//-----------------------			Inicia lavagem nas linhas						-----------------------//
{region "Inicio de lavagem"}
//Inicio da lavagem da linha 1
IF ComandoSalvar[84] THEN
	InsertParada(Insert:= TRUE, NomeComando:= 'INICIO LAV. L1', InsertOut=> bExecuteInsert, Comando=> sCmdInsert);
	ComandoSalvar[84] := FALSE;
END_IF	
//Inicio da lavagem da linha 2 
IF ComandoSalvar[85] THEN
	InsertParada(Insert:= TRUE, NomeComando:= 'INICIO LAV. L2', InsertOut=> bExecuteInsert, Comando=> sCmdInsert);
	ComandoSalvar[85] := FALSE;
END_IF
//Inicio da lavagem da linha 3
IF ComandoSalvar[86] THEN
	InsertParada(Insert:= TRUE, NomeComando:= 'INICIO LAV. L3', InsertOut=> bExecuteInsert, Comando=> sCmdInsert);
	ComandoSalvar[86] := FALSE;
END_IF	 
//Inicio da lavagem da linha 4
IF ComandoSalvar[87] THEN
	InsertParada(Insert:= TRUE, NomeComando:= 'INICIO LAV. L4', InsertOut=> bExecuteInsert, Comando=> sCmdInsert);
	ComandoSalvar[87] := FALSE;
END_IF	 
//Inicio da lavagem da linha 5
IF ComandoSalvar[88] THEN
	InsertParada(Insert:= TRUE, NomeComando:= 'INICIO LAV. L5', InsertOut=> bExecuteInsert, Comando=> sCmdInsert);
	ComandoSalvar[88] := FALSE;
END_IF	 
//Inicio da lavagem da linha 6
IF ComandoSalvar[89] THEN
	InsertParada(Insert:= TRUE, NomeComando:= 'INICIO LAV. L6', InsertOut=> bExecuteInsert, Comando=> sCmdInsert);
	ComandoSalvar[89] := FALSE;
END_IF	 
//Inicio da lavagem da linha 7
IF ComandoSalvar[90] THEN
	InsertParada(Insert:= TRUE, NomeComando:= 'INICIO LAV. L7', InsertOut=> bExecuteInsert, Comando=> sCmdInsert);
	ComandoSalvar[90] := FALSE;
END_IF	 
//Inicio da lavagem da linha 8
IF ComandoSalvar[91] THEN
	InsertParada(Insert:= TRUE, NomeComando:= 'INICIO LAV. L8', InsertOut=> bExecuteInsert, Comando=> sCmdInsert);
	ComandoSalvar[91] := FALSE;
END_IF
//Inicio da lavagem da linha 9
IF ComandoSalvar[92] THEN
	InsertParada(Insert:= TRUE, NomeComando:= 'INICIO LAV. L9', InsertOut=> bExecuteInsert, Comando=> sCmdInsert);
	ComandoSalvar[92] := FALSE;
END_IF 
//Inicio da lavagem da linha 10
IF ComandoSalvar[93] THEN
	InsertParada(Insert:= TRUE, NomeComando:= 'INICIO LAV. L10', InsertOut=> bExecuteInsert, Comando=> sCmdInsert);
	ComandoSalvar[93] := FALSE;
END_IF
//Inicio da lavagem da linha 11
IF ComandoSalvar[94] THEN
	InsertParada(Insert:= TRUE, NomeComando:= 'INICIO LAV. L11', InsertOut=> bExecuteInsert, Comando=> sCmdInsert);
	ComandoSalvar[94] := FALSE;
END_IF
//Inicio da lavagem da linha 12
IF ComandoSalvar[95] THEN
	InsertParada(Insert:= TRUE, NomeComando:= 'INICIO LAV. L12', InsertOut=> bExecuteInsert, Comando=> sCmdInsert);
	ComandoSalvar[95] := FALSE;
END_IF
{endregion}

//-----------------------			Para lavagem nas linhas							-----------------------//
{Region "Para a lavagem"}
//Parada da lavagem da linha 1
IF ComandoSalvar[96] THEN
	InsertParada(Insert:= TRUE, NomeComando:= 'PARA LAV. L1', InsertOut=> bExecuteInsert, Comando=> sCmdInsert);
	ComandoSalvar[96] := FALSE;
END_IF	
//Parada da lavagem da linha 2
IF ComandoSalvar[97] THEN
	InsertParada(Insert:= TRUE, NomeComando:= 'PARA LAV. L2', InsertOut=> bExecuteInsert, Comando=> sCmdInsert);
	ComandoSalvar[97] := FALSE;
END_IF	
//Parada da lavagem da linha 3
IF ComandoSalvar[98] THEN
	InsertParada(Insert:= TRUE, NomeComando:= 'PARA LAV. L3', InsertOut=> bExecuteInsert, Comando=> sCmdInsert);
	ComandoSalvar[98] := FALSE;
END_IF	
//Parada da lavagem da linha 4
IF ComandoSalvar[99] THEN
	InsertParada(Insert:= TRUE, NomeComando:= 'PARA LAV. L4', InsertOut=> bExecuteInsert, Comando=> sCmdInsert);
	ComandoSalvar[99] := FALSE;
END_IF	
//Parada da lavagem da linha 5
IF ComandoSalvar[100] THEN
	InsertParada(Insert:= TRUE, NomeComando:= 'PARA LAV. L5', InsertOut=> bExecuteInsert, Comando=> sCmdInsert);
	ComandoSalvar[100] := FALSE;
END_IF	
//Parada da lavagem da linha 6
IF ComandoSalvar[101] THEN
	InsertParada(Insert:= TRUE, NomeComando:= 'PARA LAV. L6', InsertOut=> bExecuteInsert, Comando=> sCmdInsert);
	ComandoSalvar[101] := FALSE;
END_IF	
//Parada da lavagem da linha 7
IF ComandoSalvar[102] THEN
	InsertParada(Insert:= TRUE, NomeComando:= 'PARA LAV. L7', InsertOut=> bExecuteInsert, Comando=> sCmdInsert);
	ComandoSalvar[102] := FALSE;
END_IF	
//Parada da lavagem da linha 8
IF ComandoSalvar[103] THEN
	InsertParada(Insert:= TRUE, NomeComando:= 'PARA LAV. L8', InsertOut=> bExecuteInsert, Comando=> sCmdInsert);
	ComandoSalvar[103] := FALSE;
END_IF	
//Parada da lavagem da linha 9
IF ComandoSalvar[104] THEN
	InsertParada(Insert:= TRUE, NomeComando:= 'PARA LAV. L9', InsertOut=> bExecuteInsert, Comando=> sCmdInsert);
	ComandoSalvar[104] := FALSE;
END_IF	
//Parada da lavagem da linha 10
IF ComandoSalvar[105] THEN
	InsertParada(Insert:= TRUE, NomeComando:= 'PARA LAV. L10', InsertOut=> bExecuteInsert, Comando=> sCmdInsert);
	ComandoSalvar[105] := FALSE;
END_IF	
//Parada da lavagem da linha 11
IF ComandoSalvar[106] THEN
	InsertParada(Insert:= TRUE, NomeComando:= 'PARA LAV. L11', InsertOut=> bExecuteInsert, Comando=> sCmdInsert);
	ComandoSalvar[106] := FALSE;
END_IF	
//Parada da lavagem da linha 12
IF ComandoSalvar[107] THEN
	InsertParada(Insert:= TRUE, NomeComando:= 'PARA LAV. L12', InsertOut=> bExecuteInsert, Comando=> sCmdInsert);
	ComandoSalvar[107] := FALSE;
END_IF	
{endregion}

//-----------------------			Acionamento manual dos elevadores				-----------------------//
{Region "Acionamento Elevadores"}
//Acionamento manual do elevador 1
IF ComandoSalvar[108] THEN
	InsertParada(Insert:= TRUE, NomeComando:= 'ACION. MANUAL ELEV1', InsertOut=> bExecuteInsert, Comando=> sCmdInsert);
	ComandoSalvar[108] := FALSE;
END_IF	
//Acionamento manual do elevador 2
IF ComandoSalvar[109] THEN
	InsertParada(Insert:= TRUE, NomeComando:= 'ACION. MANUAL ELEV2', InsertOut=> bExecuteInsert, Comando=> sCmdInsert);
	ComandoSalvar[109] := FALSE;
END_IF
//Acionamento manual do elevador 3
IF ComandoSalvar[110] THEN
	InsertParada(Insert:= TRUE, NomeComando:= 'ACION. MANUAL ELEV3', InsertOut=> bExecuteInsert, Comando=> sCmdInsert);
	ComandoSalvar[110] := FALSE;
END_IF
{endregion}
	 

//-----------------------			Descargas										-----------------------//
{Region "Descargas"}
//Caixa de recebimento
IF ComandoSalvar[111] THEN
	InsertParada(Insert:= TRUE, NomeComando:= 'ACION. MANUAL CX. RECEB.', InsertOut=> bExecuteInsert, Comando=> sCmdInsert);
	ComandoSalvar[111] := FALSE;
END_IF
//Caixa de 30Ton
IF ComandoSalvar[112] THEN
	InsertParada(Insert:= TRUE, NomeComando:= 'ACION. MANUAL CX. 30TON', InsertOut=> bExecuteInsert, Comando=> sCmdInsert);
	ComandoSalvar[112] := FALSE;
END_IF
//Caixa superior
IF ComandoSalvar[113] THEN
	InsertParada(Insert:= TRUE, NomeComando:= 'ACION. MANUAL CX. SUPERIOR', InsertOut=> bExecuteInsert, Comando=> sCmdInsert);
	ComandoSalvar[113] := FALSE;
END_IF
{endregion}
	 
	 

//-----------------------			Comandos das receitas							-----------------------//
{Region "Comandos das receitas"}
//Salvar
IF ComandoSalvar[114] THEN
	InsertParada(Insert:= TRUE, NomeComando:= 'SALVAR RECEITA', InsertOut=> bExecuteInsert, Comando=> sCmdInsert);
	ComandoSalvar[114] := FALSE;
END_IF
//Carregar
IF ComandoSalvar[115] THEN
	InsertParada(Insert:= TRUE, NomeComando:= 'CARREGAR RECEITA', InsertOut=> bExecuteInsert, Comando=> sCmdInsert);
	ComandoSalvar[115] := FALSE;
END_IF
//Excluir
IF ComandoSalvar[116] THEN
	InsertParada(Insert:= TRUE, NomeComando:= 'EXCLUIR RECEITA', InsertOut=> bExecuteInsert, Comando=> sCmdInsert);
	ComandoSalvar[116] := FALSE;
END_IF
{endregion}

//-----------------------			Confirmação dos alarmes							-----------------------//
{Region "Comandos da balança"}
//Confirma alarmes
IF ComandoSalvar[117] THEN
	InsertParada(Insert:= TRUE, NomeComando:= 'CONFIRMAR ALARMES', InsertOut=> bExecuteInsert, Comando=> sCmdInsert);
	ComandoSalvar[117] := FALSE;
END_IF

//-----------------------			Comandos da balança			-----------------------//
//Confirma alarmes
IF ComandoSalvar[117] THEN
	InsertParada(Insert:= TRUE, NomeComando:= 'CORTE GROSSO', InsertOut=> bExecuteInsert, Comando=> sCmdInsert);
	ComandoSalvar[117] := FALSE;
END_IF
//Confirma alarmes
IF ComandoSalvar[117] THEN
	InsertParada(Insert:= TRUE, NomeComando:= 'CORTE FINO', InsertOut=> bExecuteInsert, Comando=> sCmdInsert);
	ComandoSalvar[117] := FALSE;
END_IF
//Confirma alarmes
IF ComandoSalvar[117] THEN
	InsertParada(Insert:= TRUE, NomeComando:= 'PESO PADRÃO', InsertOut=> bExecuteInsert, Comando=> sCmdInsert);
	ComandoSalvar[117] := FALSE;
END_IF
//Confirma alarmes
IF ComandoSalvar[117] THEN
	InsertParada(Insert:= TRUE, NomeComando:= 'CONFIRMAR ALARMES', InsertOut=> bExecuteInsert, Comando=> sCmdInsert);
	ComandoSalvar[117] := FALSE;
END_IF
{endregion}

//-----------------------			Misturador							-----------------------//
{Region "Misturador"}
//Soprador
IF ComandoSalvar[118] THEN
	InsertParada(Insert:= TRUE, NomeComando:= 'SOPRADOR MANUAL', InsertOut=> bExecuteInsert, Comando=> sCmdInsert);
	ComandoSalvar[118] := FALSE;
END_IF
	//Prato
IF ComandoSalvar[119] THEN
	InsertParada(Insert:= TRUE, NomeComando:= 'PRATO MANUAL', InsertOut=> bExecuteInsert, Comando=> sCmdInsert);
	ComandoSalvar[119] := FALSE;
END_IF
//Aspersor
IF ComandoSalvar[120] THEN
	InsertParada(Insert:= TRUE, NomeComando:= 'ASPERSOR MANUAL', InsertOut=> bExecuteInsert, Comando=> sCmdInsert);
	ComandoSalvar[120] := FALSE;
END_IF
//Descarga
IF ComandoSalvar[121] THEN
	InsertParada(Insert:= TRUE, NomeComando:= 'DESCARGA TRAT. MANUAL', InsertOut=> bExecuteInsert, Comando=> sCmdInsert);
	ComandoSalvar[121] := FALSE;
END_IF
{endregion}

END_PROGRAM

// ---- POUs/Testes Thiago/InsertBD_Comandos.TcPOU
FUNCTION_BLOCK InsertBD_Comandos
VAR_INPUT
	Insert:BOOL;	//Comando para inserir os dados
	NomeComando:STRING;	//Nome do comando
	
END_VAR
VAR_OUTPUT
	InsertOut:BOOL;
	Comando:STRING[255];
END_VAR
VAR
	Parte1Comandos: STRING(100);
	Parte2Comandos: STRING(255);
	Parte3Comandos: STRING(255);
	sCmdInsert: STRING(255);
END_VAR

//Esse bloco é para fazer insert dos comandos no banco de dados
Parte1Comandos := 'INSERT INTO `comandos` (`comando`, `data_hora`, `usuario`, `serial_maquina`) VALUES ($'';
Parte2Comandos := CONCAT('$', CURRENT_TIMESTAMP,$'', Main.NomeUsuario);
Parte3Comandos := CONCAT('$', $'', CONCAT(Main.SerialDaMaquina, '$')'));

sCmdInsert := CONCAT(Parte1Comandos,CONCAT(NomeComando, CONCAT(Parte2Comandos, Parte3Comandos)));
Comando := sCmdInsert;
InsertOut := Insert;

END_FUNCTION_BLOCK
